FUNCTION_BLOCK FB_Blink
VAR_INPUT
	
	bStart : BOOL := FALSE;
	
END_VAR
VAR_OUTPUT
	
	bBlink : BOOL := FALSE;
	
END_VAR
VAR
	
	fbPulse : TP;

END_VAR

fbPulse(IN := bStart AND NOT fbPulse.Q, PT := T#1S);

IF (fbPulse.ET <= fbPulse.PT/2) THEN
	bBlink := FALSE;
ELSE
	bBlink := TRUE;
END_IF

END_FUNCTION_BLOCK

(* stored: Version 1.1.0.1, ProductVersion 3.1.4024.12
   POU FB_Blink: Id {5cc8f38e-c103-41e7-87da-410719122bd5}, SpecialFunc None *)
